FUNCTION_BLOCK F_RIGHT (* rightmost L characters of IN *)
  (* Standard: 61131-3; Classification: standard function of character string *)
  (* Version 0.0, 2013-04-25, 4DIAC-IDE, 4DIAC-Consortium *)
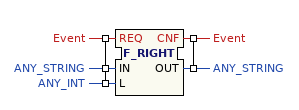
  EVENT_INPUT
    REQ WITH IN, L; (* Service Request *)
  END_EVENT
  EVENT_OUTPUT
    CNF WITH OUT; (* Confirmation of Requested Service *)
  END_EVENT
  VAR_INPUT
    IN : ANY_STRING; (* input string *)
    L : ANY_INT; (* sub-string start position *)
  END_VAR
  VAR_OUTPUT
    OUT : ANY_STRING; (* sub-string from L to string length *)
  END_VAR
END_FUNCTION_BLOCK
